FUNCTION_BLOCK PWM_control
VAR_INPUT
	dutyCycle: LREAL;
END_VAR
VAR_OUTPUT
END_VAR
VAR
END_VAR

END_FUNCTION_BLOCK

(* stored: Version 1.1.0.1, ProductVersion 3.1.4024.9
   POU PWM_control: Id {97f2005f-88d7-4913-9e3e-876430c870ed}, SpecialFunc None *)
